// TIA Portal V16 export
// export: Created 2024-12-03T15:41:39.5233176Z, ExportSetting WithDefaults, DisplayName Totally Integrated Automation Portal, DisplayVersion V16 Update 6, DisplayName TIA Portal Version Control Interface, DisplayVersion V16 Update 2, DisplayName TIA Portal Openness, DisplayVersion V16 Update 6, DisplayName TIA Portal Teamcenter Gateway, DisplayVersion V16, DisplayName SINAMICS Startdrive Advanced, DisplayVersion V16 Update 5, DisplayName SINAMICS Startdrive G130, G150, S120, S150, SINAMICS MV, S210, DisplayVersion V16 Update 5, DisplayName SINAMICS Startdrive G110M, G120, G120C, G120D, G120P, G115D, DisplayVersion V16 Update 5, DisplayName STEP 7 Professional, DisplayVersion V16 Update 6, DisplayName STEP 7 Safety, DisplayVersion V16, DisplayName WinCC Advanced / Unified PC, DisplayVersion V16 Update 6
FUNCTION_BLOCK "LightTowerGravController"   // FB34, SCL
{ S7_Optimized_Access := 'TRUE' }
VERSION : 0.1
// stored: AutoNumber true, IsIECCheckEnabled false, IsRetainMemResEnabled false, MemoryReserve 100, SetENOAutomatically false, UDAEnableTagReadback false
   VAR_INPUT
      I_full : "SmartBooldt";
      I_half_full : "SmartBooldt";
   END_VAR
   VAR_OUTPUT
      O_GREEN : Bool;
      O_ORGANGE : Bool;
      O_RED : Bool;
   END_VAR
   VAR_IN_OUT
      IO_GRAV : "Conveyor_UDT";
      IO_SUPPLY : "Conveyor_UDT";
   END_VAR
   VAR
      halfFull : TON_TIME;
      full : TON_TIME;
      empty { S7_SetPoint := 'True'} : TON_TIME;
   END_VAR
   VAR_TEMP
      T_Zone : "ZoneInfo";
      T_appstate : "ApplicationState_UDT";
   END_VAR
BEGIN
   REGION INIT

       #T_Zone := "ApplicationState_DB".ZoneNames[#IO_GRAV.Zone];
       #T_appstate := "ApplicationState_DB".Appstate[#T_Zone.AppStateIndex];

   END_REGION

   REGION Led_control

       #empty(IN := NOT #I_half_full.State AND NOT #I_full.State,
              PT := t#500ms);

       #halfFull(IN := #I_half_full.State OR #I_full.State,
                 PT := t#1s);

       #full(IN := #I_full.State AND #I_half_full.State,
             PT := t#1s);

       #IO_GRAV.Cmd.Accumulate.Acc_ext_1 := #full.Q;

       #O_RED := #full.Q;
       #O_ORGANGE := #halfFull.Q AND NOT #full.Q;
       #O_GREEN := #empty.Q;

   END_REGION

   REGION WAKE UP LANE

       IF #I_full.FE OR #I_half_full.FE THEN
           #IO_SUPPLY.Cmd.StartRequestObject := 1;
       END_IF;

   END_REGION

   REGION ALARM ACTIVE IN ZONE

       IF #T_appstate.Alarms.AlarmsActiveForHmi THEN
           #O_ORGANGE := "Clock_1Hz";
       END_IF;

   END_REGION
END_FUNCTION_BLOCK
